FUNCTION_BLOCK F_TIME_IN_US_TO_UDINT (* Convert TIME in US to UDINT *)
  (* Standard: 61499-1; Description: Copyright (c) 2023 Martin Jobst, HR Agrartechnik GmbH This program and the accompanying materials are made available under the terms of the Eclipse Public License 2.0 which is available at https://www.eclipse.org/legal/epl-2.0/ SPDX-License-Identifier: EPL-2.0 *)
  (* Version 3.0, 2025-04-14, Patrick Aigner, changed package *)
  (* Version 1.1, 2023-08-21, Franz H??pfinger, HR Agrartechnik GmbH *)
  (* Version 1.0, 2023-04-28, Martin Jobst *)
  PACKAGE iec61131::conversion;
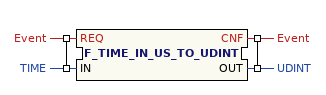
  EVENT_INPUT
    REQ WITH IN; (* Normal Execution Request *)
  END_EVENT
  EVENT_OUTPUT
    CNF WITH OUT; (* Execution Confirmation *)
  END_EVENT
  VAR_INPUT
    IN : TIME;
  END_VAR
  VAR_OUTPUT
    OUT : UDINT;
  END_VAR
  ALGORITHM REQ IN ST:
OUT := TIME_IN_US_TO_UDINT(IN);
  END_ALGORITHM
END_FUNCTION_BLOCK
